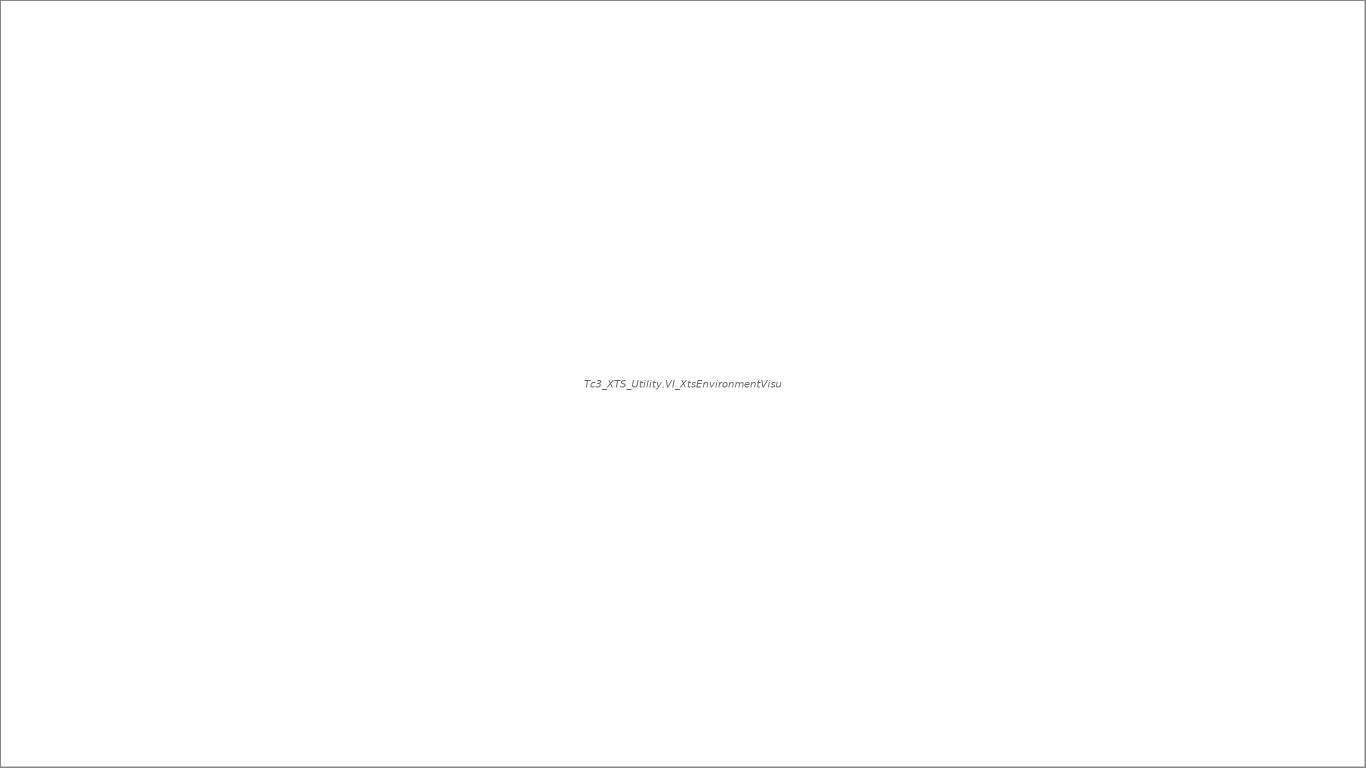
VISUALIZATION DiagnosticVisu  // 1366x768
    Frame (0,0 1366x768)
        shows Tc3_XTS_Utility.VI_XtsEnvironmentVisu()
END_VISUALIZATION

(* stored: Version 1.1.0.1
   Visu DiagnosticVisu: Id {fd3d61de-91fe-42df-b1f7-fdceb2bd410b} *)
